FUNCTION_BLOCK Switch IMPLEMENTS ITF_Cylinder
VAR_INPUT
END_VAR
VAR_OUTPUT
END_VAR
VAR
	//Hardware
	DI_Extended AT %I* : BOOL;
	DI_Retracted AT %I* : BOOL;
	DO_Extend AT %Q* : BOOL;
	//NOT USED BUT USABLE
	DI_BoundaryPressure AT %I* : BOOL;
END_VAR

PROPERTY Extended : BOOL
GET
Extended := DI_Extended;
END_GET
END_PROPERTY

METHOD METH_Extend : BOOL
DO_Extend := TRUE;
END_METHOD

METHOD METH_Retract : BOOL
DO_Extend := FALSE;
END_METHOD

PROPERTY Retracted : BOOL
GET
Retracted := DI_Retracted;
END_GET
END_PROPERTY

END_FUNCTION_BLOCK

(* stored: Version 1.1.0.1
   POU Switch: Id {fe077be6-7a16-46cf-beb7-1f9c65f24440}, SpecialFunc None
   Property Extended: Id {9e9a40d4-8f98-4c08-b532-d640e1862db4}
   Get Get: Id {a81afca2-02ea-4637-95c5-17f7143d06d5}
   Method METH_Extend: Id {421791f7-0fd8-4ba6-addf-20ea1d336999}
   Method METH_Retract: Id {bcf101fb-98a4-48e4-9d1d-e64a9673239f}
   Property Retracted: Id {8c0af0d8-f497-416f-a448-c50b38946adc}
   Get Get: Id {9dba7458-6101-48b3-9624-ab9d8211a910} *)
